TYPE st_ServiceTimeoutSetting :
STRUCT
	tRobotMovementTimeout	 : INT := 60000; // Time in ms
	tOutRobotPendingForConveyorTimeout : INT := 50000;
END_STRUCT
END_TYPE

(* stored: Version 1.1.0.1, ProductVersion 3.1.4024.13
   DUT st_ServiceTimeoutSetting: Id {ad74b4da-50fd-4d29-9164-8e6fcbaad3ff} *)
